// TIA Portal V17 export
// export: Created 2022-03-16T18:47:25.3955897Z, ExportSetting WithDefaults, DisplayName Totally Integrated Automation Portal, DisplayVersion V17, DisplayName TIA Portal Openness, DisplayVersion V17, DisplayName TIA Portal Version Control Interface, DisplayVersion V17, DisplayName STEP 7 Professional, DisplayVersion V17, DisplayName STEP 7 Safety, DisplayVersion V17, DisplayName WinCC Advanced / Unified PC, DisplayVersion V17
FUNCTION_BLOCK "EM00_00_Main"   // FB31640, LAD
TITLE = EM00_00_Main
{ S7_Optimized_Access := 'TRUE' }
AUTHOR : tech.team.motioncontrol@siemens.com
FAMILY : CPG
VERSION : 1.1
// Support: tech.team.motioncontrol@siemens.com
// stored: AutoNumber true, IsIECCheckEnabled false, IsRetainMemResEnabled false, MemoryReserve 100, SetENOAutomatically false, UDAEnableTagReadback false
   VAR
      instEventControl { ExternalAccessible := 'False'; ExternalVisible := 'False'; ExternalWritable := 'False'; S7_SetPoint := 'True'} : "EM00_01_EventControl";   // Instance DB - EM's Event Control Logic
      instPackML_ModuleSum { ExternalAccessible := 'False'; ExternalVisible := 'False'; ExternalWritable := 'False'; S7_SetPoint := 'True'} : "EM00_02_PackML_ModuleSum";   // Instance DB - EM's PackML Module Summation Logic
      instCM01 { ExternalAccessible := 'False'; ExternalVisible := 'False'; ExternalWritable := 'False'; S7_SetPoint := 'True'} : "EM00_CM01_MainOpStation";   // Instance DB - CM01
      instCM02 { ExternalAccessible := 'False'; ExternalVisible := 'False'; ExternalWritable := 'False'; S7_SetPoint := 'True'} : "EM00_CM02_Conveyor";   // Instance DB - CM02
      instCM03 { ExternalAccessible := 'False'; ExternalVisible := 'False'; ExternalWritable := 'False'; S7_SetPoint := 'True'} : "EM00_CM03_ConveyorCrossing";   // Instance DB - CM03
      instCM04 { ExternalAccessible := 'False'; ExternalVisible := 'False'; ExternalWritable := 'False'; S7_SetPoint := 'True'} : "EM00_CM04_ConveyorCrossing";   // Instance DB - CM04
      instCM05 { ExternalAccessible := 'False'; ExternalVisible := 'False'; ExternalWritable := 'False'; S7_SetPoint := 'True'} : "EM00_CM05_Conveyor";   // Instance DB - CM05
   END_VAR
   VAR_TEMP   // added for the SCL form of the ladder/FBD networks
      _w1 : Bool;
   END_VAR
BEGIN

REGION Network 1: *** BEGIN MAIN LOGIC SECTION ***
END_REGION

REGION Network 2: Call the Control Module Logic - Main Oper. Station
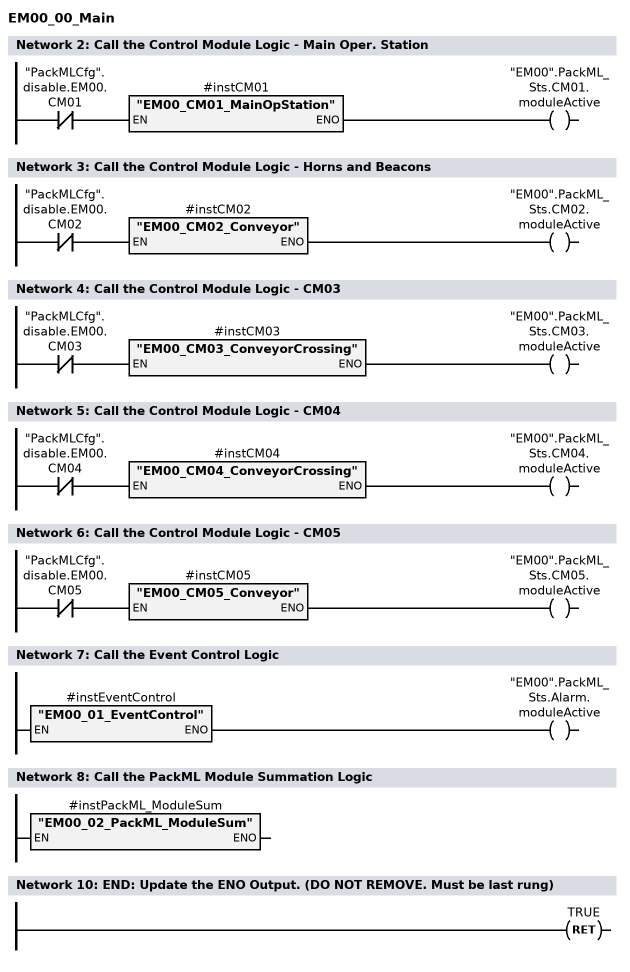
   RUNG wire#powerrail
      I_Contact( "PackMLCfg".disable.EM00.CM01 )
      #instCM01()
      Coil( "EM00".PackML_Sts.CM01.moduleActive )
   END_RUNG
   // the same network as SCL:
   #instCM01(EN := NOT "PackMLCfg".disable.EM00.CM01, ENO => #_w1);   // "EM00_CM01_MainOpStation"
   "EM00".PackML_Sts.CM01.moduleActive := #_w1;
END_REGION

REGION Network 3: Call the Control Module Logic - Horns and Beacons
   RUNG wire#powerrail
      I_Contact( "PackMLCfg".disable.EM00.CM02 )
      #instCM02()
      Coil( "EM00".PackML_Sts.CM02.moduleActive )
   END_RUNG
   // the same network as SCL:
   #instCM02(EN := NOT "PackMLCfg".disable.EM00.CM02, ENO => #_w1);   // "EM00_CM02_Conveyor"
   "EM00".PackML_Sts.CM02.moduleActive := #_w1;
END_REGION

REGION Network 4: Call the Control Module Logic - CM03
   RUNG wire#powerrail
      I_Contact( "PackMLCfg".disable.EM00.CM03 )
      #instCM03()
      Coil( "EM00".PackML_Sts.CM03.moduleActive )
   END_RUNG
   // the same network as SCL:
   #instCM03(EN := NOT "PackMLCfg".disable.EM00.CM03, ENO => #_w1);   // "EM00_CM03_ConveyorCrossing"
   "EM00".PackML_Sts.CM03.moduleActive := #_w1;
END_REGION

REGION Network 5: Call the Control Module Logic - CM04
   RUNG wire#powerrail
      I_Contact( "PackMLCfg".disable.EM00.CM04 )
      #instCM04()
      Coil( "EM00".PackML_Sts.CM04.moduleActive )
   END_RUNG
   // the same network as SCL:
   #instCM04(EN := NOT "PackMLCfg".disable.EM00.CM04, ENO => #_w1);   // "EM00_CM04_ConveyorCrossing"
   "EM00".PackML_Sts.CM04.moduleActive := #_w1;
END_REGION

REGION Network 6: Call the Control Module Logic - CM05
   RUNG wire#powerrail
      I_Contact( "PackMLCfg".disable.EM00.CM05 )
      #instCM05()
      Coil( "EM00".PackML_Sts.CM05.moduleActive )
   END_RUNG
   // the same network as SCL:
   #instCM05(EN := NOT "PackMLCfg".disable.EM00.CM05, ENO => #_w1);   // "EM00_CM05_Conveyor"
   "EM00".PackML_Sts.CM05.moduleActive := #_w1;
END_REGION

REGION Network 7: Call the Event Control Logic
   RUNG wire#powerrail
      #instEventControl()
      Coil( "EM00".PackML_Sts.Alarm.moduleActive )
   END_RUNG
   // the same network as SCL:
   #instEventControl(ENO => #_w1);   // "EM00_01_EventControl"
   "EM00".PackML_Sts.Alarm.moduleActive := #_w1;
END_REGION

REGION Network 8: Call the PackML Module Summation Logic
   RUNG wire#powerrail
      #instPackML_ModuleSum()
   END_RUNG
   // the same network as SCL:
   #instPackML_ModuleSum();   // "EM00_02_PackML_ModuleSum"
END_REGION

REGION Network 10: END: Update the ENO Output. (DO NOT REMOVE. Must be last rung)
   RUNG wire#powerrail
      ReturnCoil( TRUE )
   END_RUNG
   // the same network as SCL:
   ENO := TRUE;
   RETURN;
END_REGION
END_FUNCTION_BLOCK
